FUNCTION FUN_Multiply : REAL
VAR_INPUT
		f_Inp1			: REAL;
		f_Inp2			: REAL;
END_VAR
VAR
END_VAR

FUN_Multiply := f_Inp1 * f_Inp2;

END_FUNCTION

(* stored: Version 1.1.0.1, ProductVersion 3.1.4024.9
   POU FUN_Multiply: Id {ff1e60a7-4b2d-4678-8394-8407f996530f}, SpecialFunc None *)
